(* LS Electric XG5000 project: 241010_실습PLC와 연동 *)
(* PLC LSPLC *)

PROGRAM NewProgram (* task: 스캔 프로그램 *)
VAR
    hx00000 AT %MX0 : BOOL;
    hx00001 AT %MX1 : BOOL;
END_VAR

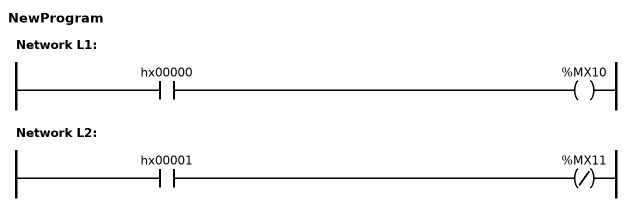
(* Rung L1 *)
%MX10 := hx00000;
(* Rung L2 *)
%MX11 := NOT hx00001;
END_PROGRAM